(* PLC project CSVExample, Beckhoff Automation GmbH TwinCAT PLC Control 3.5.13.21 *)
(* stored: creationDateTime 2022-06-19T00:13:29.5093173, modificationDateTime 2022-06-19T00:13:29.7723003 *)

FUNCTION_BLOCK CsvReader
VAR_INPUT
	en: BOOL;
	path: T_MaxString;
END_VAR
VAR_OUTPUT
	eno: BOOL := FALSE;
	err: BOOL;
	rows: UDINT;
	columns: UDINT;
END_VAR
VAR CONSTANT
	MAX_CSV_ROWS: UDINT := 1023;
	MAX_CSV_COLUMNS: UDINT := 1023;	
END_VAR
VAR	
	fbFileOpen		: FB_FileOpen;(* Opens file *)
	fbFileClose		: FB_FileClose;(* Closes file *)
	fbFileGets		: FB_FileGets;(* Reads one record (line) *)
	fbReader		: FB_CSVMemBufferReader;(* Helper function block used to parse CSV data bytes (single record line) *)

	
	line: T_MaxString;
	csv: ARRAY[0..MAX_CSV_ROWS, 0..MAX_CSV_COLUMNS] OF T_MaxString;

	
	comp_open_step: BOOL := FALSE;
	read_len: UDINT :=  0;
	n_column: UDINT := 0;
	line_parsed: BOOL := TRUE;
	comp_parse_step: BOOL := FALSE;
	comp_close_step: BOOL := FALSE;
	done: BOOL := FALSE;
END_VAR

            IF NOT en THEN
	RETURN;
END_IF

IF done THEN
	eno := TRUE;
	rows := read_len;
	columns := n_column;
	RETURN;
END_IF

(* open file step *)
IF NOT comp_open_step THEN
	fbFileOpen( sPathName := path
				, nMode := FOPEN_MODEREAD OR FOPEN_MODETEXT
				, ePath := PATH_GENERIC
				, bExecute := TRUE);
	IF fbFileOpen.bError THEN
		err := TRUE;
		RETURN;
	END_IF
	IF NOT fbFileOpen.bBusy THEN
		comp_open_step := TRUE;
	END_IF	
ELSE
	fbFileOpen(bExecute := FALSE);
END_IF

(* read line step *)
IF comp_open_step AND (NOT comp_parse_step) AND line_parsed THEN
	fbFileGets( bExecute := TRUE
				, hFile := fbFileOpen.hFile
				, sLine => line );
			
	IF fbFileGets.bError THEN
		err := FALSE;
		RETURN;
	END_IF
	IF fbFileGets.bBusy THEN
		RETURN;
	END_IF
	IF fbFileGets.bEOF OR read_len > MAX_CSV_ROWS THEN
		comp_parse_step := TRUE;
		RETURN;
	END_IF
	
	(* FB_CSVMemBufferReader needs CRLF(EOL), but FB_FileGets reaturns LF without CR. *)
	(* Thus, restore CR to before LF. *)
	IF RIGHT( line, 1 ) = '$L' THEN
		line := REPLACE( line, '$R$L', 2, LEN( line ) );
	END_IF
	
	n_column := 0;
	fbReader.eCmd := eEnumCmd_First;
	line_parsed := FALSE;
ELSE
	fbFileGets(bExecute := FALSE);
END_IF

(* parse line step *)
IF (NOT line_parsed) THEN
	fbReader( pBuffer := ADR( line ), cbBuffer := SIZEOF( line ));
	IF fbReader.bOk THEN
		fbReader.eCmd := eEnumCmd_Next;(* Read next field value *)
	
		csv[read_len, n_column] := CSVFIELD_TO_STRING(fbReader.getValue, FALSE);
		n_column := n_column + 1;
	END_IF

	IF fbReader.bCRLF OR (n_column > MAX_CSV_COLUMNS) THEN
		read_len := read_len + 1;
		line_parsed := TRUE;
	END_IF
END_IF

(* close file step *)
IF comp_parse_step AND (NOT comp_close_step) THEN
	fbFileClose( sNetId := '', hFile := fbFileOpen.hFile, bExecute := TRUE );
	
	IF fbFileClose.bError THEN
		err := TRUE;
		RETURN;
	END_IF
	IF NOT fbFileClose.bBusy THEN
		comp_close_step := TRUE;
	END_IF
ELSE
	fbFileClose(bExecute := FALSE);	
END_IF
		
IF comp_close_step THEN
	done := TRUE;
END_IF
          

METHOD Get : T_MaxString
VAR_INPUT
	en: BOOL;
	col: UDINT;
	row: UDINT;
END_VAR
                  IF NOT en THEN
	RETURN;
END_IF

IF (col <= MAX_CSV_COLUMNS) AND (col <= MAX_CSV_ROWS) THEN
	Get := csv[col, row];
END_IF
                
END_METHOD
END_FUNCTION_BLOCK
